// TIA Portal V21 export
TYPE "coneCrusherOut"
   STRUCT
      sgStart : Bool;
      sgStop : Bool;
      preStartAlmOn : Bool;
      feedEn : Bool;   // Allow feed from upstream unit
   END_STRUCT;
END_TYPE
